// TIA Portal V18 export
TYPE "UDT_AHUSetpoints"
// stored: IsFailsafeCompliant false
   STRUCT
      Room : Struct
         Actual { S7_SetPoint := 'True'} : "UDT_SetPointsBasic";
         Target { S7_SetPoint := 'True'} : "UDT_SetPointsBasic";
         Shift { S7_SetPoint := 'True'} : "UDT_SetPointsBasic";
      END_STRUCT;
      Supply { S7_SetPoint := 'True'} : "UDT_AHUsSATSetPoints";
   END_STRUCT;
   // Room.Shift.RATHeating[1..2] := 0.0;
   // Room.Shift.RATCooling[1..2] := 0.0;
   // Room.Shift.IAQ[1..2] := 0.0;
   // Room.Shift.BuildingdP[1..2] := 0.0;
END_TYPE
